{attribute 'OPC.UA.DA.JobMethod' := 'JobMethode_CuttingProcess'}
FUNCTION_BLOCK MBS_MR02_AS_CuttingProcess
VAR
	AlwaysTrue : BOOL := TRUE;
	// Used for debugging purposes to display InputArguments of method call
	MethodCall_CuttingProcess : BOOL := FALSE; // used to store InputArg "MethodCall" from Start() method
	ProcessingTime_CuttingProcess : TIME;
	TS_EndschalterEntlastung : BOOL;
	callCounterStart : ULINT; // counts how many times the Start() method has been called
	callCounterCheckState : ULINT; // counts how many times the CheckState() method has been called
	callCounterAbort : ULINT; // counts how many times the Abort() method has been called
	
	// Variables to determine if a job has been started (Start() method has been called) or finished
	jobRunning : BOOL;
	jobFinished : BOOL;

	// State machine variable
	state : UDINT;
	
	//Variablen des FBs
	ResetCall : BOOL;
	MBS_MR02_CuttingProcess : CuttingProcess;
END_VAR
	
VAR_INPUT
	NotAusSignal: BOOL;
	LightSensor_01 : BOOL;
END_VAR

VAR_OUTPUT
	CuttingMaschine_Ansteuerung : BOOL;
END_VAR

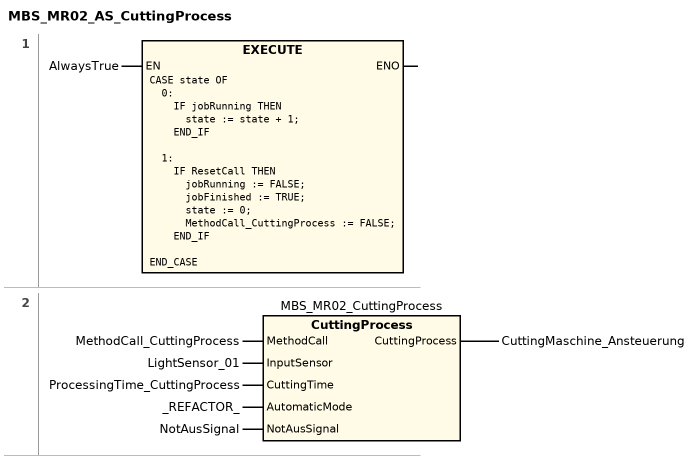
// NETWORK 1
IF AlwaysTrue THEN
    CASE state OF
    	0:
    		IF jobRunning THEN
    			state := state + 1;
    		END_IF
    		
    	1:
    		IF ResetCall THEN
    			jobRunning := FALSE;
    			jobFinished := TRUE;
    			state := 0;
    			MethodCall_CuttingProcess := FALSE;
    		END_IF
    		
    END_CASE
END_IF

// NETWORK 2
MBS_MR02_CuttingProcess(
    MethodCall := MethodCall_CuttingProcess,
    InputSensor := LightSensor_01,
    CuttingTime := ProcessingTime_CuttingProcess,
    AutomaticMode := _REFACTOR_,
    NotAusSignal := NotAusSignal); // CuttingProcess
CuttingMaschine_Ansteuerung := MBS_MR02_CuttingProcess.CuttingProcess;

{attribute 'TcRpcEnable' := '1'}
METHOD Abort : HRESULT
VAR_INPUT
	hdl : UDINT; // Do not change, used by server.
END_VAR
callCounterAbort := callCounterAbort + 1;
END_METHOD

{attribute 'TcRpcEnable' := '1'}
METHOD CheckState : HRESULT
VAR_INPUT
	hdl : UDINT; // Do not change, used by server.
END_VAR
VAR_OUTPUT
	bBusy : BOOL; // Do not change. Used by server to find out if the job is finished
	
	// List of OutputArguments for OPC UA method, may be customized
	State : BOOL; // Abgeschlossener MethodCall
	MethodCall: BOOL; //Input Recall
END_VAR
callCounterCheckState := callCounterCheckState + 1;
IF NOT jobFinished THEN
	bBusy := TRUE; // job is not finished yet
	CheckState := 0; // no error
ELSE
	bBusy := FALSE; // job is finished
	CheckState := 0; // done, no error occured during execution (OPC UA StatusCode "GOOD")
	jobFinished := FALSE;
	State := ResetCall;
	MethodCall := MethodCall_CuttingProcess;
END_IF
END_METHOD

{attribute 'TcRpcEnable' := '1'}
METHOD Start : HRESULT
VAR_INPUT
	// List of InputArguments for OPC UA method, may be customized
	MethodCall : BOOL; // some description
	ProcessingTime : TIME;
END_VAR
VAR_OUTPUT
	hdl : UDINT; // Do not change, used by server.
END_VAR
callCounterStart := callCounterStart + 1;

MethodCall_CuttingProcess := MethodCall;
ProcessingTime_CuttingProcess := ProcessingTime;

jobRunning := TRUE;
Start := 0; // no error occured, e.g. while parsing the input arguments (0 = OPC UA StatusCode "GOOD")
END_METHOD

END_FUNCTION_BLOCK

(* stored: Version 1.1.0.1, ProductVersion 3.1.4024.15
   POU MBS_MR02_AS_CuttingProcess: Id {2d7d64da-63fe-4e9c-ab0f-e6acdd3925d6}, SpecialFunc None
   Method Abort: Id {80b3a94c-bcbb-42ae-99e5-0c65da5ec65c}
   Method CheckState: Id {9b40824c-1d23-4dfb-a644-afed068e893f}
   Method Start: Id {919cd498-2f6d-4e31-ab0e-fc58556f06d1} *)
